FUNCTION_BLOCK sequence_B_08_AX_AX (* Sequence with 8 Outputs, Transition by BOOL level, with AX Adapter *)
  (* Standard: 61499-2; Description: Copyright (c) 2026 HR Agrartechnik GmbH This program and the accompanying materials are made available under the terms of the Eclipse Public License 2.0 which is available at https://www.eclipse.org/legal/epl-2.0/ SPDX-License-Identifier: EPL-2.0 *)
  (* Version 1.0, 2026-04-20, Franz Höpfinger, HR Agrartechnik GmbH, initial API and implementation - Level based transitions for power-fail recovery *)
  PACKAGE logiBUS::utils::sequence::bool;
  IMPORT eclipse4diac::core::TypeHash;
  IMPORT logiBUS::utils::sequence::const::sequence;
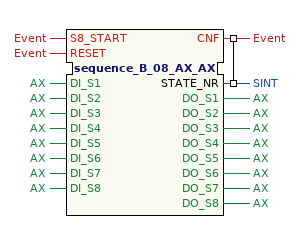
  EVENT_INPUT
    S8_START; (* jump from State_08 to START *)
    RESET; (* Reset from any State to START *)
  END_EVENT
  EVENT_OUTPUT
    CNF WITH STATE_NR; (* Execution Confirmation *)
  END_EVENT
  VAR_OUTPUT
    STATE_NR : SINT; (* State Number, START = 0, State_01 = 1 and so on. *)
  END_VAR
  SOCKETS
    DI_S1 : adapter::types::unidirectional::AX; (* jump from START to State_01 *)
    DI_S2 : adapter::types::unidirectional::AX; (* jump from State_01 to State_02 *)
    DI_S3 : adapter::types::unidirectional::AX; (* jump from State_02 to State_03 *)
    DI_S4 : adapter::types::unidirectional::AX; (* jump from State_03 to State_04 *)
    DI_S5 : adapter::types::unidirectional::AX; (* jump from State_04 to State_05 *)
    DI_S6 : adapter::types::unidirectional::AX; (* jump from State_05 to State_06 *)
    DI_S7 : adapter::types::unidirectional::AX; (* jump from State_06 to State_07 *)
    DI_S8 : adapter::types::unidirectional::AX; (* jump from State_07 to State_08 *)
  END_SOCKETS
  PLUGS
    DO_S1 : adapter::types::unidirectional::AX; (* Output if State_01 is active *)
    DO_S2 : adapter::types::unidirectional::AX; (* Output if State_02 is active *)
    DO_S3 : adapter::types::unidirectional::AX; (* Output if State_03 is active *)
    DO_S4 : adapter::types::unidirectional::AX; (* Output if State_04 is active *)
    DO_S5 : adapter::types::unidirectional::AX; (* Output if State_05 is active *)
    DO_S6 : adapter::types::unidirectional::AX; (* Output if State_06 is active *)
    DO_S7 : adapter::types::unidirectional::AX; (* Output if State_07 is active *)
    DO_S8 : adapter::types::unidirectional::AX; (* Output if State_08 is active *)
  END_PLUGS
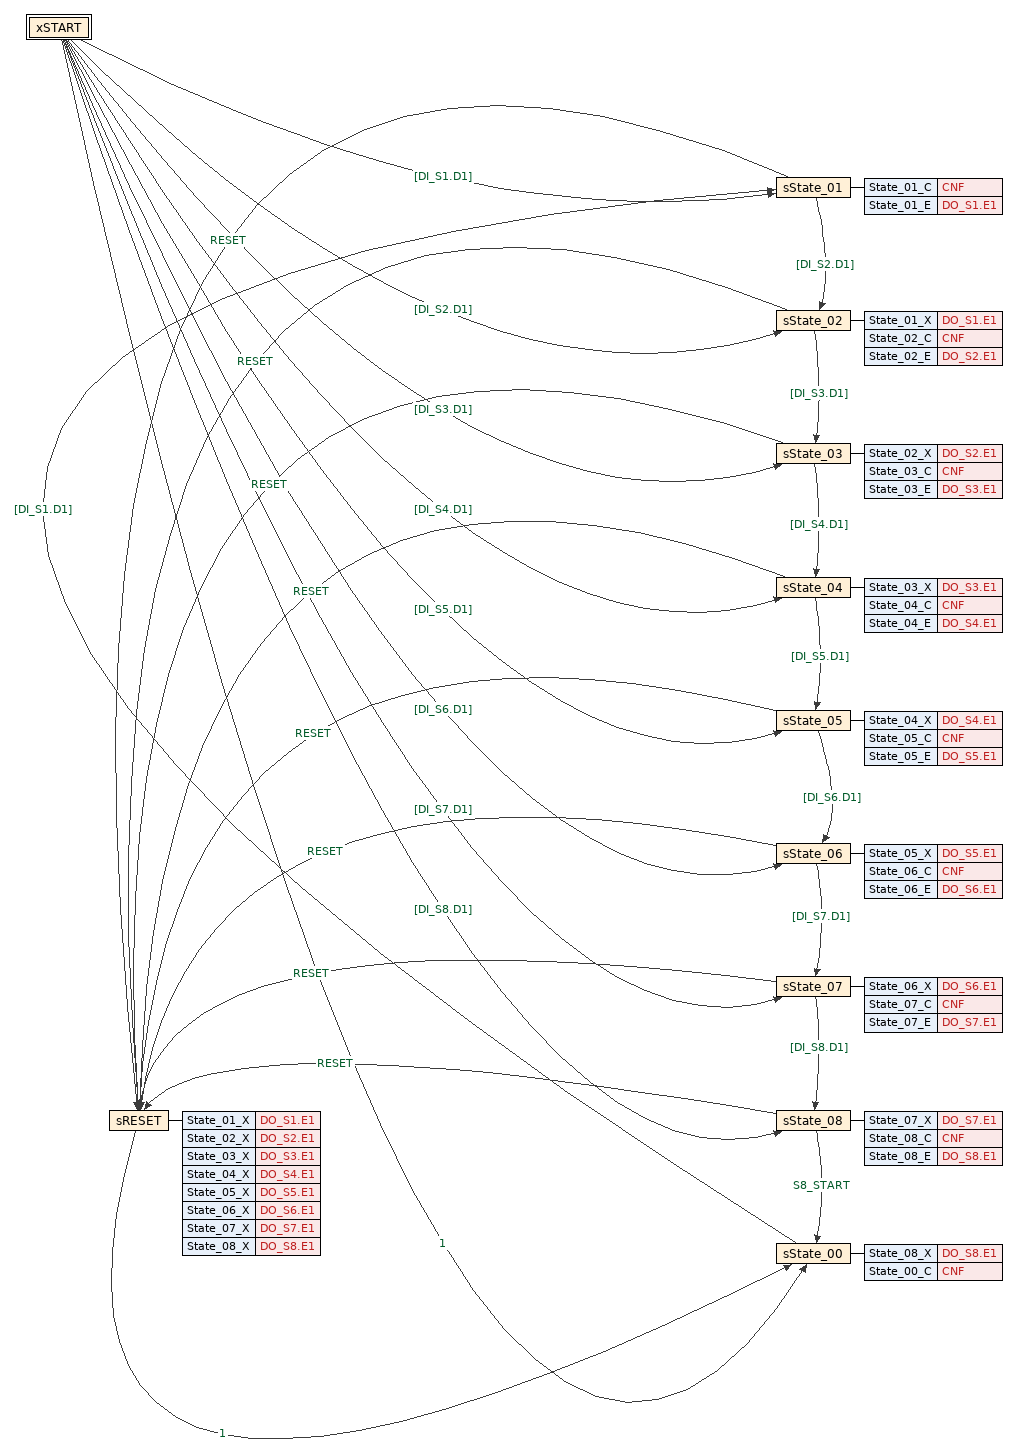
  EC_STATES
    xSTART; (* Initial State *)
    sState_01 : State_01_C -> CNF, State_01_E -> DO_S1.E1;
    sState_02 : State_01_X -> DO_S1.E1, State_02_C -> CNF, State_02_E -> DO_S2.E1;
    sState_03 : State_02_X -> DO_S2.E1, State_03_C -> CNF, State_03_E -> DO_S3.E1;
    sState_04 : State_03_X -> DO_S3.E1, State_04_C -> CNF, State_04_E -> DO_S4.E1;
    sState_05 : State_04_X -> DO_S4.E1, State_05_C -> CNF, State_05_E -> DO_S5.E1;
    sState_06 : State_05_X -> DO_S5.E1, State_06_C -> CNF, State_06_E -> DO_S6.E1;
    sState_07 : State_06_X -> DO_S6.E1, State_07_C -> CNF, State_07_E -> DO_S7.E1;
    sState_08 : State_07_X -> DO_S7.E1, State_08_C -> CNF, State_08_E -> DO_S8.E1;
    sState_00 : State_08_X -> DO_S8.E1, State_00_C -> CNF;
    sRESET : State_01_X -> DO_S1.E1, State_02_X -> DO_S2.E1, State_03_X -> DO_S3.E1, State_04_X -> DO_S4.E1, State_05_X -> DO_S5.E1, State_06_X -> DO_S6.E1, State_07_X -> DO_S7.E1, State_08_X -> DO_S8.E1;
  END_STATES
  EC_TRANSITIONS
    xSTART TO sState_08 := [DI_S8.D1]; (* Recovery logic *)
    xSTART TO sState_07 := [DI_S7.D1]; (* Recovery logic *)
    xSTART TO sState_06 := [DI_S6.D1]; (* Recovery logic *)
    xSTART TO sState_05 := [DI_S5.D1]; (* Recovery logic *)
    xSTART TO sState_04 := [DI_S4.D1]; (* Recovery logic *)
    xSTART TO sState_03 := [DI_S3.D1]; (* Recovery logic *)
    xSTART TO sState_02 := [DI_S2.D1]; (* Recovery logic *)
    xSTART TO sState_01 := [DI_S1.D1]; (* Recovery logic *)
    xSTART TO sState_00 := 1;
    sState_00 TO sState_01 := [DI_S1.D1];
    sState_01 TO sState_02 := [DI_S2.D1];
    sState_02 TO sState_03 := [DI_S3.D1];
    sState_03 TO sState_04 := [DI_S4.D1];
    sState_04 TO sState_05 := [DI_S5.D1];
    sState_05 TO sState_06 := [DI_S6.D1];
    sState_06 TO sState_07 := [DI_S7.D1];
    sState_07 TO sState_08 := [DI_S8.D1];
    sState_08 TO sState_00 := S8_START; (* Loop back remains event-driven or can be changed *)
    sState_01 TO sRESET := RESET;
    sState_02 TO sRESET := RESET;
    sState_03 TO sRESET := RESET;
    sState_04 TO sRESET := RESET;
    sState_05 TO sRESET := RESET;
    sState_06 TO sRESET := RESET;
    sState_07 TO sRESET := RESET;
    sState_08 TO sRESET := RESET;
    sRESET TO sState_00 := 1;
  END_TRANSITIONS
  ALGORITHM State_00_C IN ST:
STATE_NR := sequence::State_00;
  END_ALGORITHM
  ALGORITHM State_01_C IN ST:
STATE_NR := sequence::State_01;
  END_ALGORITHM
  ALGORITHM State_02_C IN ST:
STATE_NR := sequence::State_02;
  END_ALGORITHM
  ALGORITHM State_03_C IN ST:
STATE_NR := sequence::State_03;
  END_ALGORITHM
  ALGORITHM State_04_C IN ST:
STATE_NR := sequence::State_04;
  END_ALGORITHM
  ALGORITHM State_05_C IN ST:
STATE_NR := sequence::State_05;
  END_ALGORITHM
  ALGORITHM State_06_C IN ST:
STATE_NR := sequence::State_06;
  END_ALGORITHM
  ALGORITHM State_07_C IN ST:
STATE_NR := sequence::State_07;
  END_ALGORITHM
  ALGORITHM State_08_C IN ST:
STATE_NR := sequence::State_08;
  END_ALGORITHM
  ALGORITHM State_01_E IN ST:
DO_S1.D1 := DI_S1.D1; // ON
  END_ALGORITHM
  ALGORITHM State_01_X IN ST:
DO_S1.D1 := BOOL#FALSE;
  END_ALGORITHM
  ALGORITHM State_02_E IN ST:
DO_S2.D1 := DI_S2.D1; // ON
  END_ALGORITHM
  ALGORITHM State_02_X IN ST:
DO_S2.D1 := BOOL#FALSE;
  END_ALGORITHM
  ALGORITHM State_03_E IN ST:
DO_S3.D1 := DI_S3.D1; // ON
  END_ALGORITHM
  ALGORITHM State_03_X IN ST:
DO_S3.D1 := BOOL#FALSE;
  END_ALGORITHM
  ALGORITHM State_04_E IN ST:
DO_S4.D1 := DI_S4.D1; // ON
  END_ALGORITHM
  ALGORITHM State_04_X IN ST:
DO_S4.D1 := BOOL#FALSE;
  END_ALGORITHM
  ALGORITHM State_05_E IN ST:
DO_S5.D1 := DI_S5.D1; // ON
  END_ALGORITHM
  ALGORITHM State_05_X IN ST:
DO_S5.D1 := BOOL#FALSE;
  END_ALGORITHM
  ALGORITHM State_06_E IN ST:
DO_S6.D1 := DI_S6.D1; // ON
  END_ALGORITHM
  ALGORITHM State_06_X IN ST:
DO_S6.D1 := BOOL#FALSE;
  END_ALGORITHM
  ALGORITHM State_07_E IN ST:
DO_S7.D1 := DI_S7.D1; // ON
  END_ALGORITHM
  ALGORITHM State_07_X IN ST:
DO_S7.D1 := BOOL#FALSE;
  END_ALGORITHM
  ALGORITHM State_08_E IN ST:
DO_S8.D1 := DI_S8.D1; // ON
  END_ALGORITHM
  ALGORITHM State_08_X IN ST:
DO_S8.D1 := BOOL#FALSE;
  END_ALGORITHM
END_FUNCTION_BLOCK
